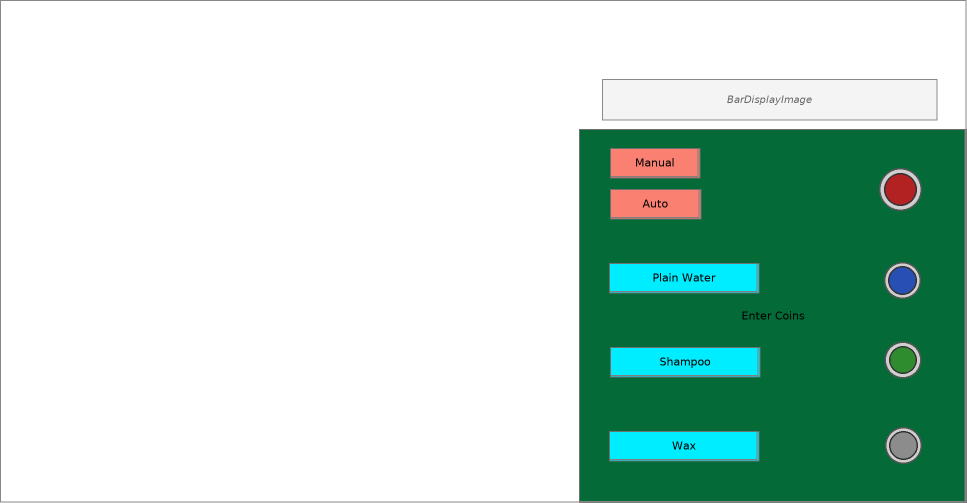
VISUALIZATION Visualization  // 967x503
    Button (579,129 388x374), "Enter Coins", invisible if: MAIN.bCoinEnter
        toggle MAIN.bCoinEnter
    Group (609,257 317x210), invisible if: NOT MAIN.bAuto AND NOT MAIN.bManual
        Button (0,6 150x30), "Plain Water", input disabled if: MAIN.bAuto
            toggle MAIN.bPlainWater
        Button (1,90 150x30), "Shampoo", input disabled if: MAIN.bAuto
            toggle MAIN.bShampoo
        Button (0,174 150x30), "Wax", input disabled if: MAIN.bAuto
            toggle MAIN.bWax
        Lamp1 (272,0 43x47), variable: MAIN.bLedW, style: Lamp-Lamp1-Blue
        Lamp1 (271,82 46x42), variable: MAIN.bLedS, style: Lamp-Lamp1-Green
        Lamp1 (272,167 45x43), variable: MAIN.bLedWx, style: Lamp-Lamp1-Gray
    Group (602,79 335x140), invisible if: NOT MAIN.bCoinEnter
        BarDisplayImage (0,0 335x41), value: MAIN.tTimer.ET, style: BarDisplayImage-Gray, scale format: %.1f, scale 0..20000
        Button (8,69 90x30), "Manual", invisible if: MAIN.bAuto
            toggle MAIN.bManual
        Button (8,110 91x30), "Auto", invisible if: MAIN.bManual
            toggle MAIN.bAuto
        Lamp1 (274,82 49x57), variable: MAIN.bLedPower, style: Lamp-Lamp1-Red
END_VISUALIZATION

(* stored: Version 1.1.0.1, ProductVersion 3.1.4024.9
   Visu Visualization: Id {11dbeaa3-a4c0-4f2e-8abe-680c95b1d14d} *)
